// Mitsubishi GX Works2 project: 241108_PLC_STUDY2   PLC: Q02U

PROGRAM MAIN
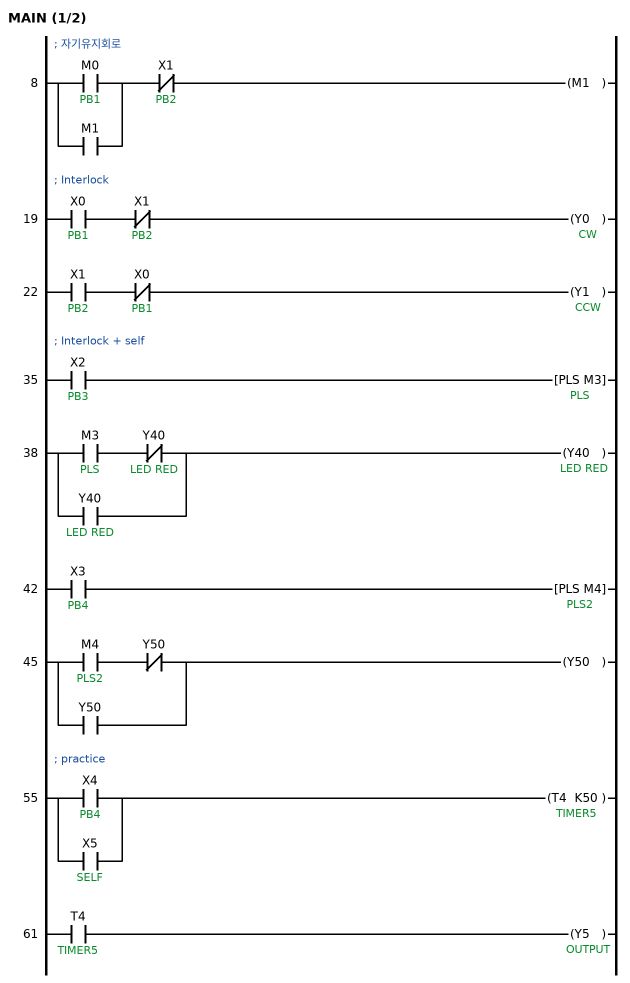
; 자기유지회로
8     LD      M0  ; PB1
      OR      M1
      ANI     X1  ; PB2
      OUT     M1
; Interlock
19    LD      X0  ; PB1
      ANI     X1  ; PB2
      OUT     Y0  ; CW
22    LD      X1  ; PB2
      ANI     X0  ; PB1
      OUT     Y1  ; CCW
; Interlock + self
35    LD      X2  ; PB3
      PLS     M3  ; PLS
38    LD      M3  ; PLS
      ANI     Y40  ; LED RED
      OR      Y40  ; LED RED
      OUT     Y40  ; LED RED
42    LD      X3  ; PB4
      PLS     M4  ; PLS2
45    LD      M4  ; PLS2
      ANI     Y50
      OR      Y50
      OUT     Y50
; practice
55    LD      X4  ; PB4
      OR      X5  ; SELF
      OUT     T4 K50  ; TIMER5
61    LD      T4  ; TIMER5
      OUT     Y5  ; OUTPUT
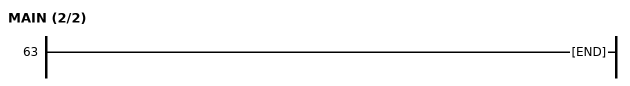
63    END
END_PROGRAM

// device comments not shown above
Y4  ; FALL
